Staubli VAL3: encodeJoint.pgx

program encodeJoint(joint& value, num& buffer[])
  local num elements[6]
begin
  elements[0] = value.j1
  elements[1] = value.j2
  elements[2] = value.j3
  elements[3] = value.j4
  elements[4] = value.j5
  elements[5] = value.j6

  toBinary(elements, 6, "4.0b", buffer)
end
